PROGRAM MAIN
VAR
END_VAR

END_PROGRAM

(* stored: Version 1.1.0.1, ProductVersion 3.1.0.38
   POU MAIN: Id {40038b9a-d30f-400b-a531-eb7ec579e2c4}, SpecialFunc None *)
